TYPE structAnalysis :
STRUCT
	axis:typeDataAxis; //the data itself
	box1:structBoxData;
	box2:structBoxData;
	box3:structBoxData;
END_STRUCT
END_TYPE

(* stored: Version 1.1.0.1, ProductVersion 3.1.4024.11
   DUT structAnalysis: Id {20351ee5-43ff-0162-31c8-c1d76145921f} *)
